// TIA Portal V17 export
// export: Created 2022-07-20T07:01:27.1570389Z, ExportSetting WithDefaults, DisplayName Totally Integrated Automation Portal, DisplayVersion V17, DisplayName TIA Portal Openness, DisplayVersion V17, DisplayName TIA Portal Version Control Interface, DisplayVersion V17, DisplayName SINAMICS Startdrive Advanced, DisplayVersion V17, DisplayName SINAMICS Startdrive G130, G150, S120, S150, SINAMICS MV, S210, DisplayVersion V17, DisplayName SINAMICS Startdrive G110M, G120, G120C, G120D, G120P, G115D, DisplayVersion V17, DisplayName STEP 7 Professional, DisplayVersion V17, DisplayName STEP 7 Safety, DisplayVersion V17, DisplayName WinCC Advanced, DisplayVersion V17
FUNCTION_BLOCK "FB10260_AisScannerManager"   // FB10260, LAD
{ S7_Optimized_Access := 'TRUE' }
VERSION : 0.1
// stored: AutoNumber false, IsIECCheckEnabled false, IsRetainMemResEnabled false, MemoryReserve 100, SetENOAutomatically false, UDAEnableTagReadback false
   VAR_INPUT
      AisScannerActivatedSensor : Bool;
      RequestAisScannerActivation : Bool;
   END_VAR
   VAR_OUTPUT
      ActivateAisScanner : Bool;
      AisScannerActivated : Bool;
   END_VAR
BEGIN

REGION Network 1 (SCL): First Scan
   IF "FirstScan" THEN
       ;
   END_IF;
END_REGION

REGION Network 2 (SCL): Ais Scanner Management
   IF #RequestAisScannerActivation THEN
       #ActivateAisScanner := TRUE;
   ELSE
       #ActivateAisScanner := FALSE;
   END_IF;
END_REGION

REGION Network 3 (SCL): Ais Scanner States Management
   #AisScannerActivated := NOT (#AisScannerActivatedSensor);
END_REGION
END_FUNCTION_BLOCK
